// TwinCAT 3 PLC project Autonomous_Cart
// ProgramVersion: 3.1.4023.0
// libraries:
//   Tc2_Standard, * (Beckhoff Automation GmbH)
//   Tc2_System, * (Beckhoff Automation GmbH)
//   Tc3_Module, * (Beckhoff Automation GmbH)
// project tree:
//   / PlcTask.TcTTO
//   POUs/ MAIN.TcPOU
// real-time tasks:
//   TASK PlcTask: cycle T#10ms, priority 20, ADS port 350
// I/O:
//   DEVICE Device 1 (EtherCAT), AmsNetId 10.95.1.7.2.1
//     Head unit(EK1100) [EK1100 EtherCAT Coupler (2A E-Bus)]
//       Safety PLC [EL6900, TwinSAFE PLC]
//       Safety In [EL1904, 4 Ch. Safety Input 24V, TwinSAFE]
//         modules: Module 1 (FSOES)
//       analog output (EL4002) [EL4002 2Ch. Ana. Output 0-10V, 12bit]
//       analog input (EL3062) [EL3062 2Ch. Ana. Input 0-10V]
// variable links:
//   Device 1 (EtherCAT) <-> Device 1 (EtherCAT)/Head unit(EK1100)/Safety In
//     Head unit(EK1100)/Safety PLC/ConnectionInputs/Message_2 TxPDO <-> Module 1 (FSOES)/RxPDO/FSOE
//   Device 1 (EtherCAT) <-> Device 1 (EtherCAT)/Head unit(EK1100)/Safety PLC
//     Head unit(EK1100)/Safety In/Module 1 (FSOES)/TxPDO/FSOE <-> ConnectionOutputs/Message_2 RxPDO

CONFIGURATION Autonomous_Cart
    RESOURCE PLC ON TwinCAT3
        TASK PlcTask(INTERVAL := T#10ms, PRIORITY := 20);
        PROGRAM MAIN WITH PlcTask : MAIN;
    END_RESOURCE
END_CONFIGURATION

// ---- POUs/MAIN.TcPOU
PROGRAM MAIN
VAR
	CurrentNum AT%IB10:INT;
	CurrentVoltage : REAL;
	
	Overname : BOOL;
	Autonoom : BOOL;
	AutonomousButton : BOOL;
END_VAR

IF Autonoom THEN
	CurrentVoltage := CurrentNum/6552;
	Autonoom R= CurrentVoltage > 1;
END_IF
Autonoom S= AutonomousButton;

END_PROGRAM
